FUNCTION_BLOCK SS3_Lid_feeder (* Basic FB with empty ECC *)
  (* Standard: 61499-2 *)
  (* Version 1.0, 2025-08-24, DEVIASH *)
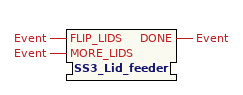
  EVENT_INPUT
    FLIP_LIDS;
    MORE_LIDS;
  END_EVENT
  EVENT_OUTPUT
    DONE;
  END_EVENT
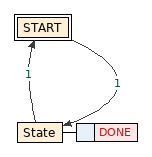
  EC_STATES
    START; (* Initial State *)
    State : -> DONE;
  END_STATES
  EC_TRANSITIONS
    START TO State := 1;
    State TO START := 1;
  END_TRANSITIONS
END_FUNCTION_BLOCK
